ABB RobotStudio station: Solution initial test.rsstn

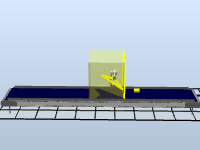
Station Solution1 (saved by RobotStudio 6.8.8148.134)
Controller System1, task T_ROB1: task frame (RAPID world) sits at (5535.63, 748.67, 709.58) mm in the station
Controller System1
  mechanical unit ROB_1: IRB1600_10_145__01, 6 joints, base frame (480.91, -394.38, -359.58) mm, rotated rx 0 ry 0 rz 90 deg
  mechanical unit CNV1: ?, 1 joints, base frame (0, 0, 0) mm
Layout (positions relative to the parent item):
  - bin mover_3 [smart component, from libraries\bin mover.rslib] at (-500, 0, 0) mm
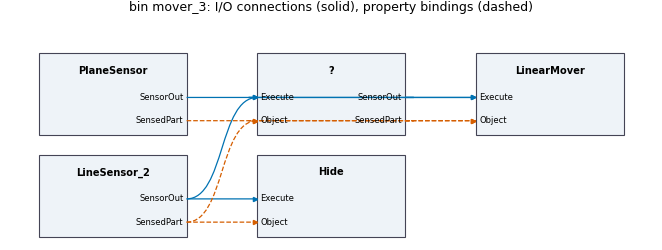
      connections:
        ?.SensorOut -> LinearMover.Execute
        PlaneSensor.SensorOut -> LinearMover.Execute
        ?.SensorOut -> ?.Execute
        LineSensor_2.SensorOut -> ?.Execute
        LineSensor_2.SensorOut -> Hide.Execute
        ?.SensedPart => LinearMover.Object
        PlaneSensor.SensedPart => LinearMover.Object
        ?.SensedPart => ?.Object
        LineSensor_2.SensedPart => ?.Object
        LineSensor_2.SensedPart => Hide.Object
    - LinearMover [smart component, from Components\LinearMover.rslib] at (6663.26, 677.27, 1050.93) mm, rotated rx 180 ry 0 rz 90 deg
        properties: Object=(none); Direction=[0 0 -1]; Speed=8; Reference=Global; ReferenceObject=(none)
    - PlaneSensor [smart component, from Components\PlaneSensor.rslib]
        properties: Origin=[7.419145 0.146999 1.42]; Axis1=[0 0 -1.35]; Axis2=[0 0.4 0]; SensedPart=(none)
      - _sensorPart_ [part, from libraries\bin mover.rslib]
    - LineSensor_2 [smart component, from Components\LineSensor.rslib]
        properties: Start=[7.369145 0.346999 0.008]; End=[7.369145 0.346999 0.123]; Radius=0.09; SensedPart=(none); SensedPoint=[0 0 0]
      - _sensorPart_ [part, from libraries\bin mover.rslib]
    - Hide [smart component, from Components\Hide.rslib]
        properties: Object=(none)
  - bin1_2 [part, from libraries\bin1.rslib] at (6733.74, 347, -12) mm
  - conveyor 1 [part] at (0, -1500, -4460) mm, rotated rx 90 ry 0 rz 90 deg
  - Suction gripper 18cm [smart component] at (6016.55, 985.44, 1386.5) mm, rotated rx -180 ry 0 rz -90 deg
      signals: DI do1
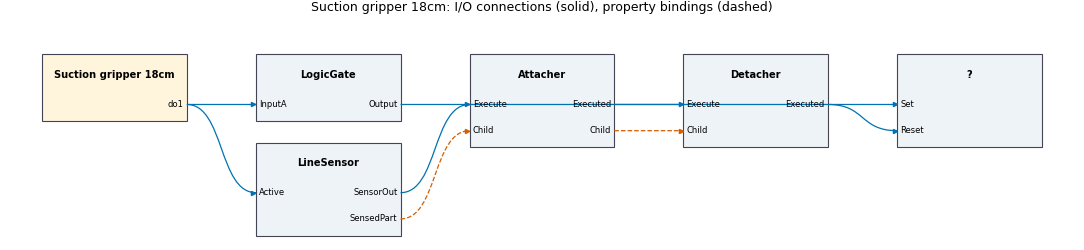
      connections:
        Suction gripper 18cm.do1 -> LogicGate.InputA
        Suction gripper 18cm.do1 -> LineSensor.Active
        LogicGate.Output -> Detacher.Execute
        LineSensor.SensorOut -> Attacher.Execute
        Attacher.Executed -> ?.Set
        Detacher.Executed -> ?.Reset
        LineSensor.SensedPart => Attacher.Child
        Attacher.Child => Detacher.Child
    - Attacher [smart component, from Components\Attacher.rslib]
        properties: Parent=Suction_gripper 18cm; Flange=0; Child=Yellow block; Mount=false; Offset=[0 0 0]; Orientation=[0 0 0]
    - LogicGate [smart component, from Components\LogicGate.rslib]
        properties: Operator=NOT; Delay=0
    - LineSensor [smart component, from Components\LineSensor.rslib] at (7150.29, 306.47, 1168.39) mm, rotated rx 180 ry 0 rz 90 deg
        properties: Start=[-0.30577796087058 -7.14894421240012 1.16938863540814]; End=[-0.305777964813962 -7.14894420825673 1.13938863540814]; Radius=0.09; SensedPart=Yellow block; SensedPoint=[6.7271533203125 0.417008178710937 1.3712216796875]
      - _sensorPart_ [part]
    - Detacher [smart component, from Components\Detacher.rslib]
        properties: Child=Yellow block; KeepPosition=true
  - Suction_gripper 18cm [mechanism, from libraries\Suction_gripper_18cm.rslib] at (6016.55, 985.44, 1471.5) mm, rotated rx -180 ry 0 rz -90 deg
  - IRB1600_10_145__01 [mechanism, from Robots\IRB1600_10_145_G_01.rslib] at (6016.55, 235.44, 350) mm, rotated rx 0 ry 0 rz 90 deg; joint values [0, 0, 0, 0, 1.5708, 0] (rad or m)
  - 输送链 [conveyor]
    - Conveyor cover [part] at (-300, 0, 14) mm
    - Yellow block [part] at (0, -475.41, 0) mm
    - 传送带对象_40 [conveyorobject] at (10403.63, 748.67, 709.58) mm
      - Yellow block [part] at (-415.92, -1776.06, -1501.58) mm
    - 传送带对象_41 [conveyorobject] at (7703.63, 748.67, 709.58) mm
      - Yellow block [part] at (-391.49, -1776.41, -1499.83) mm
    - 传送带对象_42 [conveyorobject] at (5003.63, 748.67, 709.58) mm
      - Yellow block [part] at (-394.03, -1778.07, -1491.94) mm
    - 传送带对象_43 [conveyorobject] at (2303.63, 748.67, 709.58) mm
      - Yellow block [part] at (-500, -1095, -698) mm
Attachment: Suction gripper 18cm is attached to Suction_gripper 18cm / Suction gripper 18cm
Attachment: Suction_gripper 18cm is attached to IRB1600_10_145__01 / Link6
Conveyor tracking 连接_2: unit CNV1, TravelOffset=3.7, QueueTrackDistance=0, StartWindowWidth=1.8, SyncSeparation=0, CountsPerMeter=10000
Station logic (signal -> signal, property => property):
  System1.do_attach -> Suction gripper 18cm.do1
Targets, tools, work objects and paths stored in the station, written as RAPID:
! task T_ROB1
MODULE CalibData
  PERS tooldata Suction_gripper_18cm:=[TRUE,[[0,0,85],[1,0,0,0]],[1,[0,0,1],[1,0,0,0],0,0,0]];
  TASK PERS wobjdata wobj_cnv1:=[FALSE,FALSE,"CNV1",[[0,0,0],[1,0,0,0]],[[0,0,0],[1,0,0,0]]];
ENDMODULE

! task T_ROB1
MODULE Module1
  CONST robtarget Target_10:=[[480.915,236.77,676.92],[0,-0.707106781,0.707106781,0],[0,0,0,0],[9E+09,9E+09,9E+09,9E+09,9E+09,0]];
  CONST robtarget Target_20:=[[29.699626144,355.874016057,111.58001204],[0.000000002,0.707106781,-0.707106781,0.000000007],[0,-1,0,0],[9E+09,9E+09,9E+09,9E+09,9E+09,0]];
  CONST robtarget Target_30:=[[1192.207950487,-330.312717415,676.919992598],[0.000000021,0.707106781,-0.707106781,0.000000022],[-1,-1,-1,0],[9E+09,9E+09,9E+09,9E+09,9E+09,0]];
  PROC Path_10()
    MoveL Target_10,vmax,z0,Suction_gripper_18cm\WObj:=wobj0;
    MoveL Target_20,vmax,z10,Suction_gripper_18cm\WObj:=wobj_cnv1;
    Set do_attach;
    MoveL Target_30,vmax,fine,Suction_gripper_18cm\WObj:=wobj0;
    Reset do_attach;
    MoveL Target_10,vmax,z0,Suction_gripper_18cm\WObj:=wobj0;
  ENDPROC
  PROC main()
    ActUnit CNV1;
    WaitWObj wobj_cnv1;
    Path_10;
    DropWObj wobj_cnv1;
  ENDPROC
ENDMODULE

